{attribute 'c++_compatible'}
FUNCTION_BLOCK FB_CustomTcp EXTENDS FB_SimpleTcpClient
VAR
	nRcvCnt : UDINT;
	sData : STRING(255);
END_VAR

METHOD FB_init : BOOL
VAR_INPUT
	bInitRetains : BOOL; // if TRUE, the retain variables are initialized (warm start / cold start)
	bInCopyCode : BOOL;  // if TRUE, the instance afterwards gets moved into the copy code (online change)
END_VAR
VAR
	ipSrv : ITComObjectServer;
END_VAR
sName := 'FB_CustomTcp';
sVersion := '1.0.0.0';
END_METHOD

END_FUNCTION_BLOCK

(* stored: Version 1.1.0.1, ProductVersion 3.1.4019.2
   POU FB_CustomTcp: Id {5957cace-372b-48d3-ae24-79666929e881}, SpecialFunc None
   Method FB_init: Id {78fec908-3c2e-4b31-89e3-ec846b8660da} *)
